//{attribute 'pack_mode' := '8'}
TYPE ST_ToleranceThresholdCS :
STRUCT
		GoodReadPercentagePAL		:	STRING(6);
END_STRUCT
END_TYPE

(* stored: Version 1.1.0.1
   DUT ST_ToleranceThresholdCS: Id {2ecaf75c-30ce-483b-9373-f222fdf77873} *)
